{attribute 'GeneratedUsingTerminal: EPP1004-0061-0016'}
{attribute addProperty BoxType "EPP1004-0061-0016"}
{attribute addProperty Id "InputAT %I*BOOL1"}
{attribute addProperty CRC "2198356929"}
{attribute addProperty Size "1"}
TYPE Channel_830843C1 EXTENDS InputBase_8311D824 :
STRUCT
	{attribute addProperty Name "Input"}
	Input AT %I* : BOOL;
END_STRUCT
END_TYPE

(* stored: Version 1.2.0.0, ProductVersion 3.1.4024.9
   DUT Channel_830843C1: Id {0cb393c0-ec29-4325-89fd-59923229f538} *)
